{attribute 'GeneratedUsingTerminal: EP1122-0001-0017'}
{attribute addProperty BoxType "EP1122-0001-0017"}
{attribute addProperty Id "A_0026_EP1122_0001_0018A_0026_EP1122_0001_0018_C9AEDEF81330"}
{attribute addProperty CRC "4036469690"}
{attribute addProperty Size "1330"}
TYPE A_0025_EP1122_0001_0017_F097A3BA EXTENDS EP1122_1FC0878B :
STRUCT
	{attribute addProperty Name "A_0026_EP1122_0001_0018"}
	{attribute addProperty PreviousPort "A_0025(EP1122-0001-0017) : D"}
	A_0026_EP1122_0001_0018 : A_0026_EP1122_0001_0018_C9AEDEF8;
END_STRUCT
END_TYPE

(* stored: Version 1.2.0.0, ProductVersion 3.1.4024.9
   DUT A_0025_EP1122_0001_0017_F097A3BA: Id {62dd3ed3-22bc-4041-a501-05c222e48078} *)
